VAR_GLOBAL
		stDutData_Cnc2					: ST_Dut_Data;
END_VAR

(* stored: Version 1.1.0.1, ProductVersion 3.1.4024.12
   GVL GVL_CNC2: Id {f8563509-2806-4ec9-81ec-c6d3f09f0cb0} *)
